Omron CX-Programmer project NewProject (CX-Programmer 9.61)

# PLC Pratica_avaliacao: CP1L M

## Global symbols (name address type ; comment)
0.00 BOOL  ; PB1
0.01 BOOL  ; PB2
0.02 BOOL  ; PB3
0.03 BOOL  ; SEN1
0.04 BOOL  ; SEN2
0.05 BOOL  ; LS1
0.06 BOOL  ; LS2
100.00 BOOL  ; MOP
100.01 BOOL  ; MOA
100.02 BOOL  ; MOF
200.00 BOOL  ; Etapa 0
200.01 BOOL  ; Etapa 1
200.02 BOOL  ; Etapa 2
W1.00 BOOL  ; Parado
W1.01 BOOL  ; Subir
W1.02 BOOL  ; Descer

## Program NewProgram1 (cyclic task 0)

### Section Section1

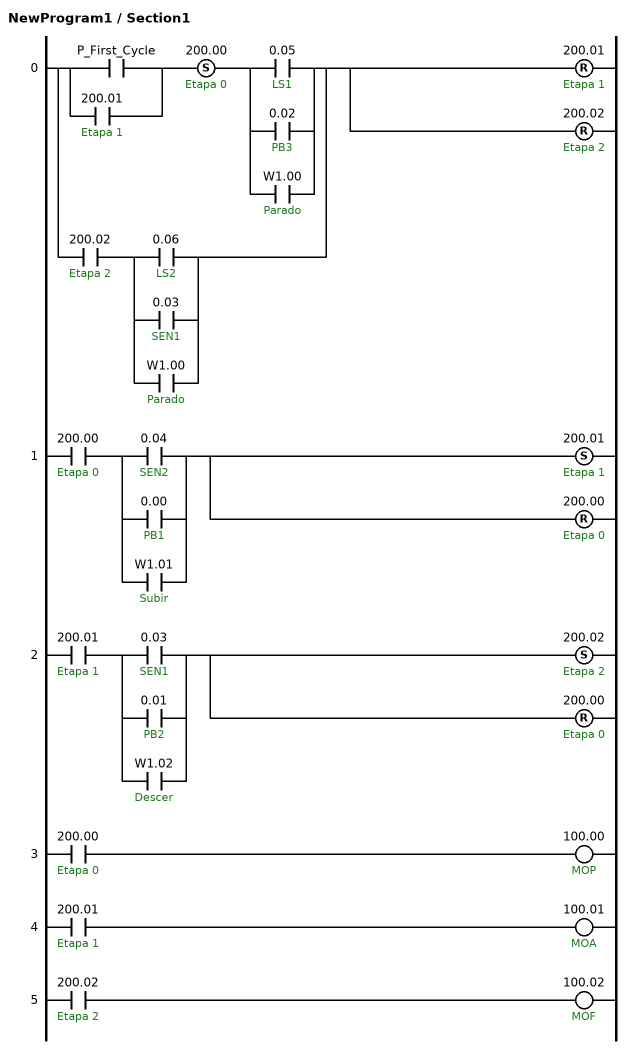
; rung 0
LD P_First_Cycle
OR 200.01  ; Etapa 1
SET 200.00  ; Etapa 0
LD 0.05  ; LS1
OR 0.02  ; PB3
OR W1.00  ; Parado
ANDLD
LD 200.02  ; Etapa 2
LD 0.06  ; LS2
OR 0.03  ; SEN1
OR W1.00  ; Parado
ANDLD
ORLD
RSET 200.01  ; Etapa 1
RSET 200.02  ; Etapa 2
; rung 1
LD 200.00  ; Etapa 0
LD 0.04  ; SEN2
OR 0.00  ; PB1
OR W1.01  ; Subir
ANDLD
SET 200.01  ; Etapa 1
RSET 200.00  ; Etapa 0
; rung 2
LD 200.01  ; Etapa 1
LD 0.03  ; SEN1
OR 0.01  ; PB2
OR W1.02  ; Descer
ANDLD
SET 200.02  ; Etapa 2
RSET 200.00  ; Etapa 0
; rung 3
LD 200.00  ; Etapa 0
OUT 100.00  ; MOP
; rung 4
LD 200.01  ; Etapa 1
OUT 100.01  ; MOA
; rung 5
LD 200.02  ; Etapa 2
OUT 100.02  ; MOF

### Section END
; rung 0
END(001)